// SIMATIC S7-200 project (STEP 7-Micro/WIN), CPU 224XP CN REL 02.02

SYMBOL_TABLE 用户定义3
一楼呼叫             I0.1     // SB1
二楼呼叫             I0.2     // SB2
三楼呼叫             I0.3     // SB3
响应一楼呼叫           Q0.1     // HL1
响应二楼呼叫           Q0.2     // HL2
响应三楼呼叫           Q0.3     // HL3
一楼响应保持           M1.1
二楼响应保持           M1.2
三楼响应保持           M1.3
电梯在一楼            Q0.4     // SQ1
电梯在二楼            Q0.5     // SQ2
电梯在三楼            Q0.6     // SQ3
开门               Q0.0
关门               Q2.1
电梯停止             Q0.7
电机正转             Q1.0     // 正在上升
电机反转             Q1.1     // 下降
上升保持             M3.2     // 电梯属于上升状态
下降保持             M3.3     // 电梯属于下降状态
楼层位置             VW0      // 数据寄存，1楼值1，2楼值2
呼叫数              VW2      // 有多少个电梯正在呼叫
上行定时器            T37      // 电梯移动时间的计数器
下行定时器            T38
开始关门             T56
停止关门             T57
门寄存器             M2.0     // 前4秒开门灯亮，第4秒关灯亮，第5秒继续运行
重置               I0.0     // 按下后电梯重置
END_SYMBOL_TABLE

ORGANIZATION_BLOCK 主程序:OB1
TITLE=程序注释
BEGIN
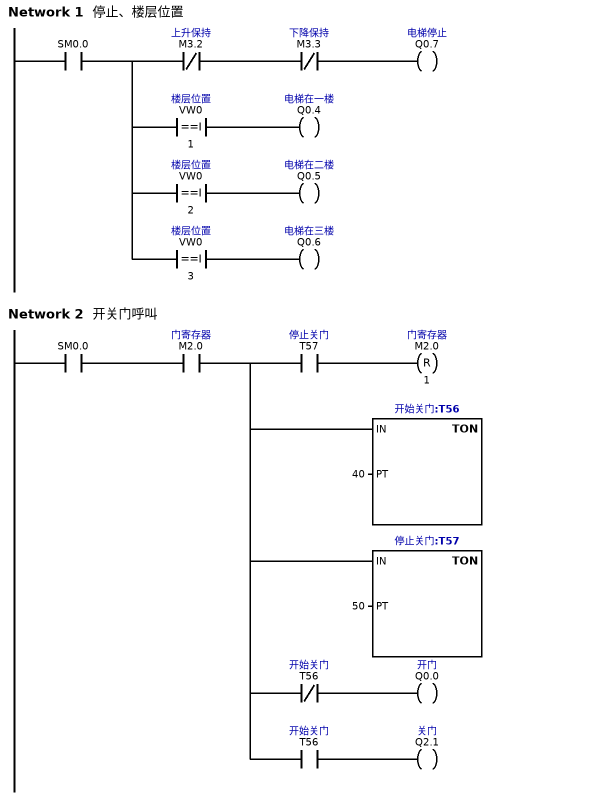
Network 1 // 停止、楼层位置
LD     SM0.0
LPS
AN     上升保持:M3.2
AN     下降保持:M3.3
=      电梯停止:Q0.7
LRD
AW=    楼层位置:VW0, 1
=      电梯在一楼:Q0.4
LRD
AW=    楼层位置:VW0, 2
=      电梯在二楼:Q0.5
LPP
AW=    楼层位置:VW0, 3
=      电梯在三楼:Q0.6
Network 2 // 开关门呼叫
LD     SM0.0
A      门寄存器:M2.0
LPS
A      停止关门:T57
R      门寄存器:M2.0, 1
LRD
TON    开始关门:T56, 40
LRD
TON    停止关门:T57, 50
LRD
AN     开始关门:T56
=      开门:Q0.0
LPP
A      开始关门:T56
=      关门:Q2.1
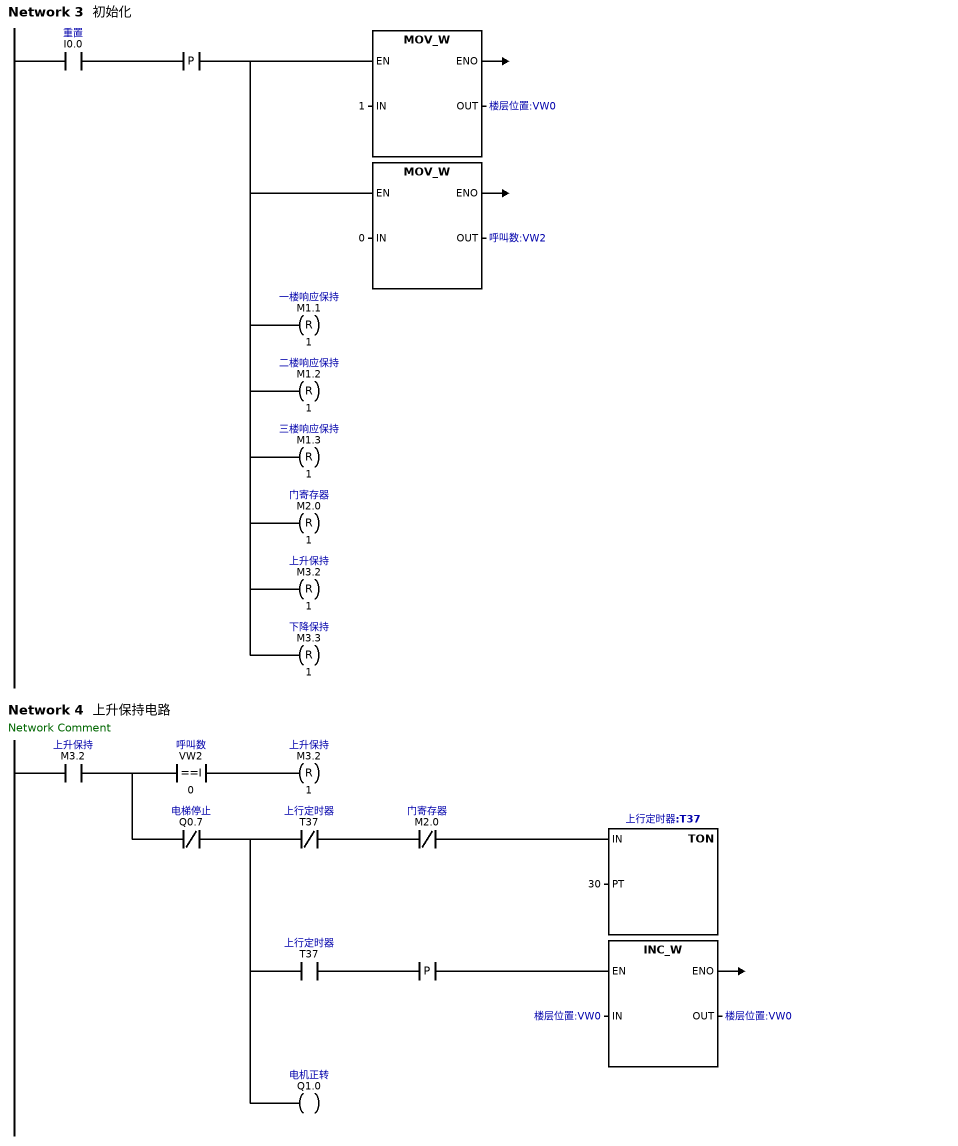
Network 3 // 初始化
LD     重置:I0.0
EU
MOVW   1, 楼层位置:VW0
MOVW   0, 呼叫数:VW2
R      一楼响应保持:M1.1, 1
R      二楼响应保持:M1.2, 1
R      三楼响应保持:M1.3, 1
R      门寄存器:M2.0, 1
R      上升保持:M3.2, 1
R      下降保持:M3.3, 1
Network 4 // 上升保持电路
// Network Comment
LD     上升保持:M3.2
LPS
AW=    呼叫数:VW2, 0
R      上升保持:M3.2, 1
LPP
AN     电梯停止:Q0.7
LPS
AN     上行定时器:T37
AN     门寄存器:M2.0
TON    上行定时器:T37, 30
LRD
A      上行定时器:T37
EU
INCW   楼层位置:VW0
LPP
=      电机正转:Q1.0
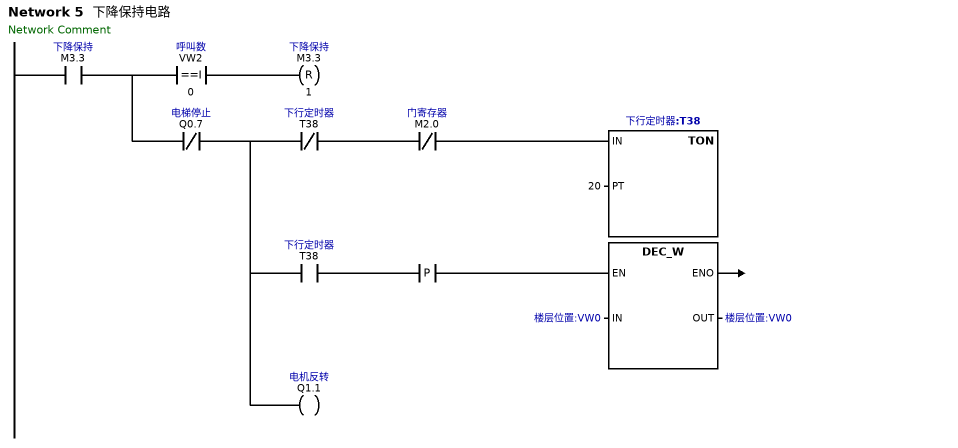
Network 5 // 下降保持电路
// Network Comment
LD     下降保持:M3.3
LPS
AW=    呼叫数:VW2, 0
R      下降保持:M3.3, 1
LPP
AN     电梯停止:Q0.7
LPS
AN     下行定时器:T38
AN     门寄存器:M2.0
TON    下行定时器:T38, 20
LRD
A      下行定时器:T38
EU
DECW   楼层位置:VW0
LPP
=      电机反转:Q1.1
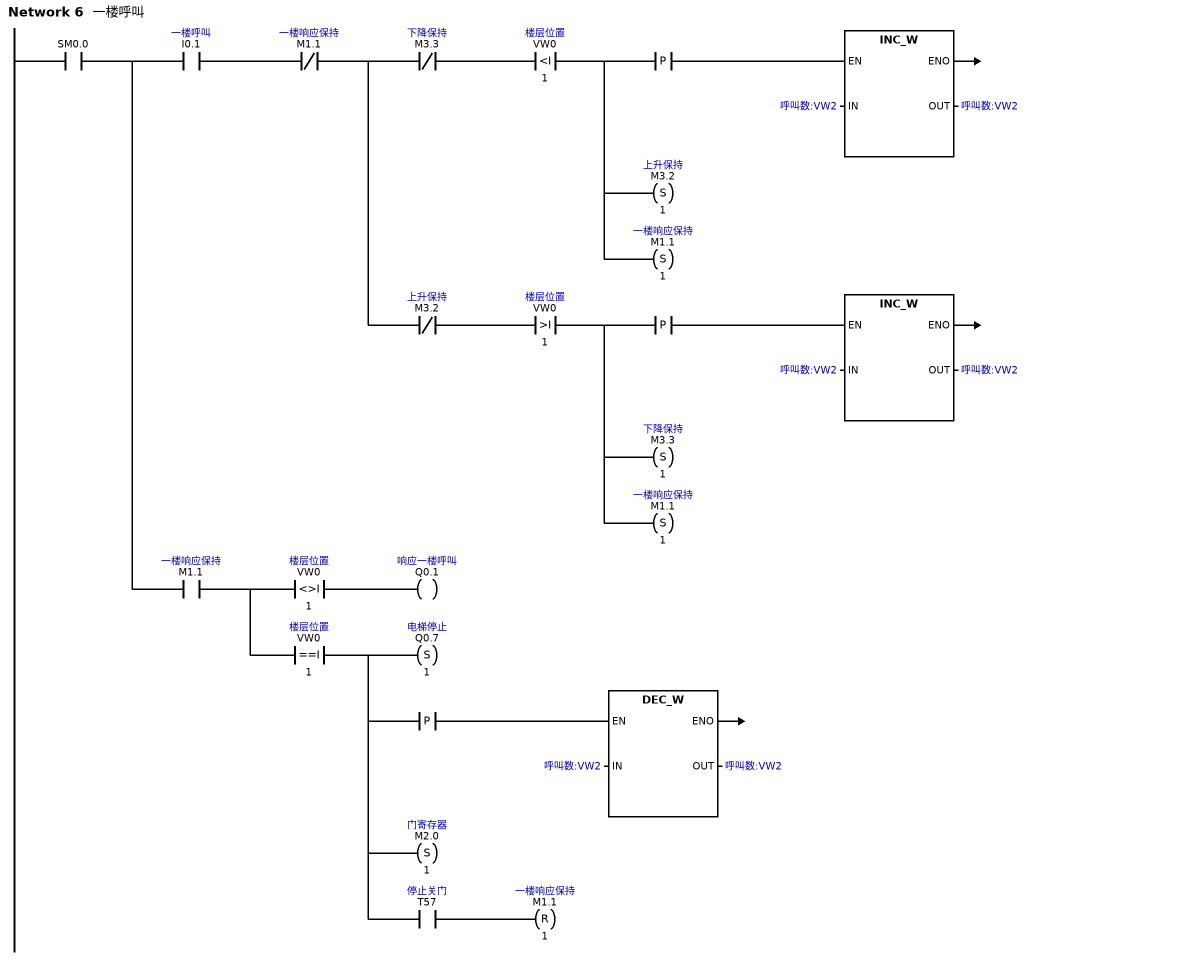
Network 6 // 一楼呼叫
LD     SM0.0
LPS
A      一楼呼叫:I0.1
AN     一楼响应保持:M1.1
LPS
AN     下降保持:M3.3
AW<    楼层位置:VW0, 1
LPS
EU
INCW   呼叫数:VW2
LRD
S      上升保持:M3.2, 1
LPP
S      一楼响应保持:M1.1, 1
LPP
AN     上升保持:M3.2
AW>    楼层位置:VW0, 1
LPS
EU
INCW   呼叫数:VW2
LRD
S      下降保持:M3.3, 1
LPP
S      一楼响应保持:M1.1, 1
LPP
A      一楼响应保持:M1.1
LPS
AW<>   楼层位置:VW0, 1
=      响应一楼呼叫:Q0.1
LPP
AW=    楼层位置:VW0, 1
LPS
S      电梯停止:Q0.7, 1
EU
DECW   呼叫数:VW2
LRD
S      门寄存器:M2.0, 1
LPP
A      停止关门:T57
R      一楼响应保持:M1.1, 1
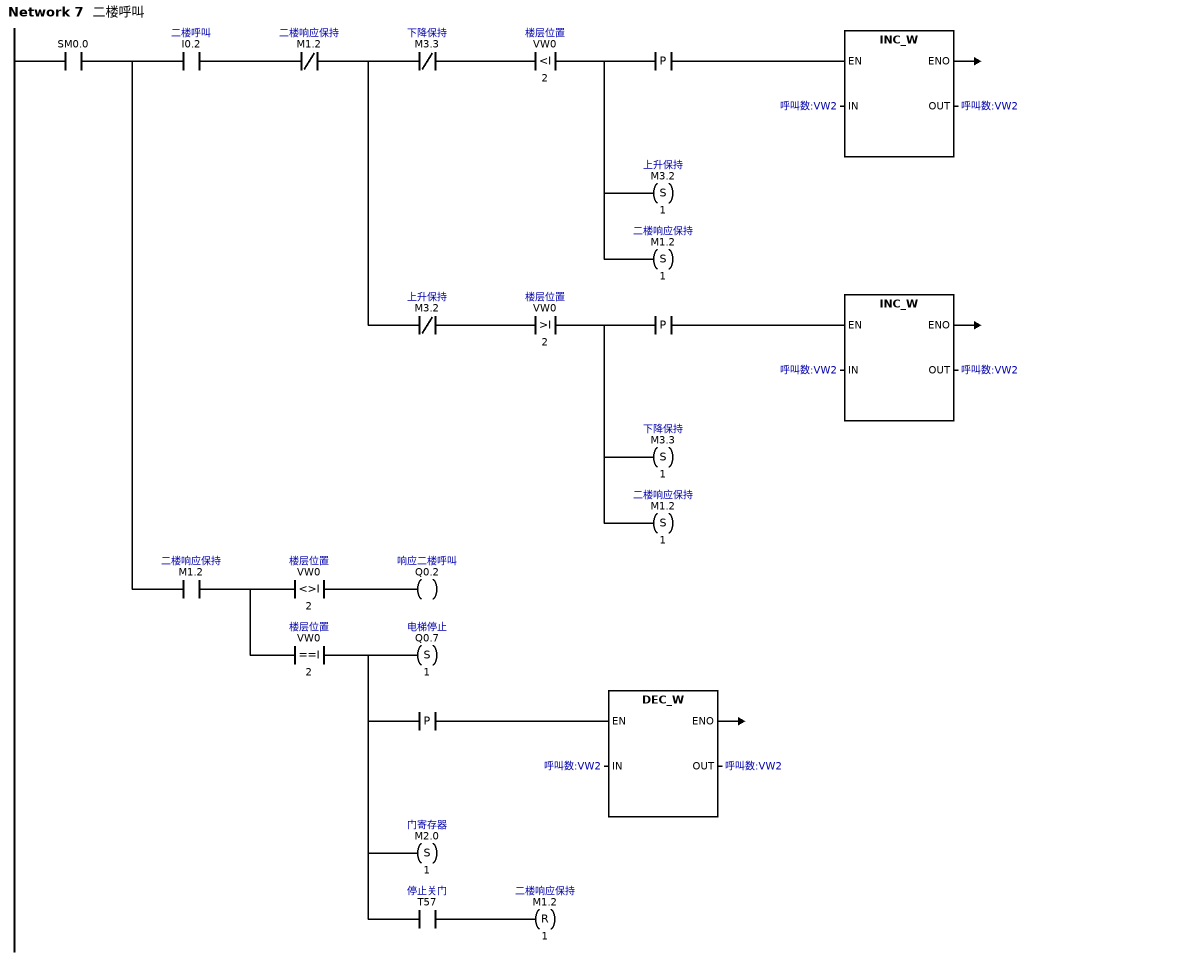
Network 7 // 二楼呼叫
LD     SM0.0
LPS
A      二楼呼叫:I0.2
AN     二楼响应保持:M1.2
LPS
AN     下降保持:M3.3
AW<    楼层位置:VW0, 2
LPS
EU
INCW   呼叫数:VW2
LRD
S      上升保持:M3.2, 1
LPP
S      二楼响应保持:M1.2, 1
LPP
AN     上升保持:M3.2
AW>    楼层位置:VW0, 2
LPS
EU
INCW   呼叫数:VW2
LRD
S      下降保持:M3.3, 1
LPP
S      二楼响应保持:M1.2, 1
LPP
A      二楼响应保持:M1.2
LPS
AW<>   楼层位置:VW0, 2
=      响应二楼呼叫:Q0.2
LPP
AW=    楼层位置:VW0, 2
LPS
S      电梯停止:Q0.7, 1
EU
DECW   呼叫数:VW2
LRD
S      门寄存器:M2.0, 1
LPP
A      停止关门:T57
R      二楼响应保持:M1.2, 1
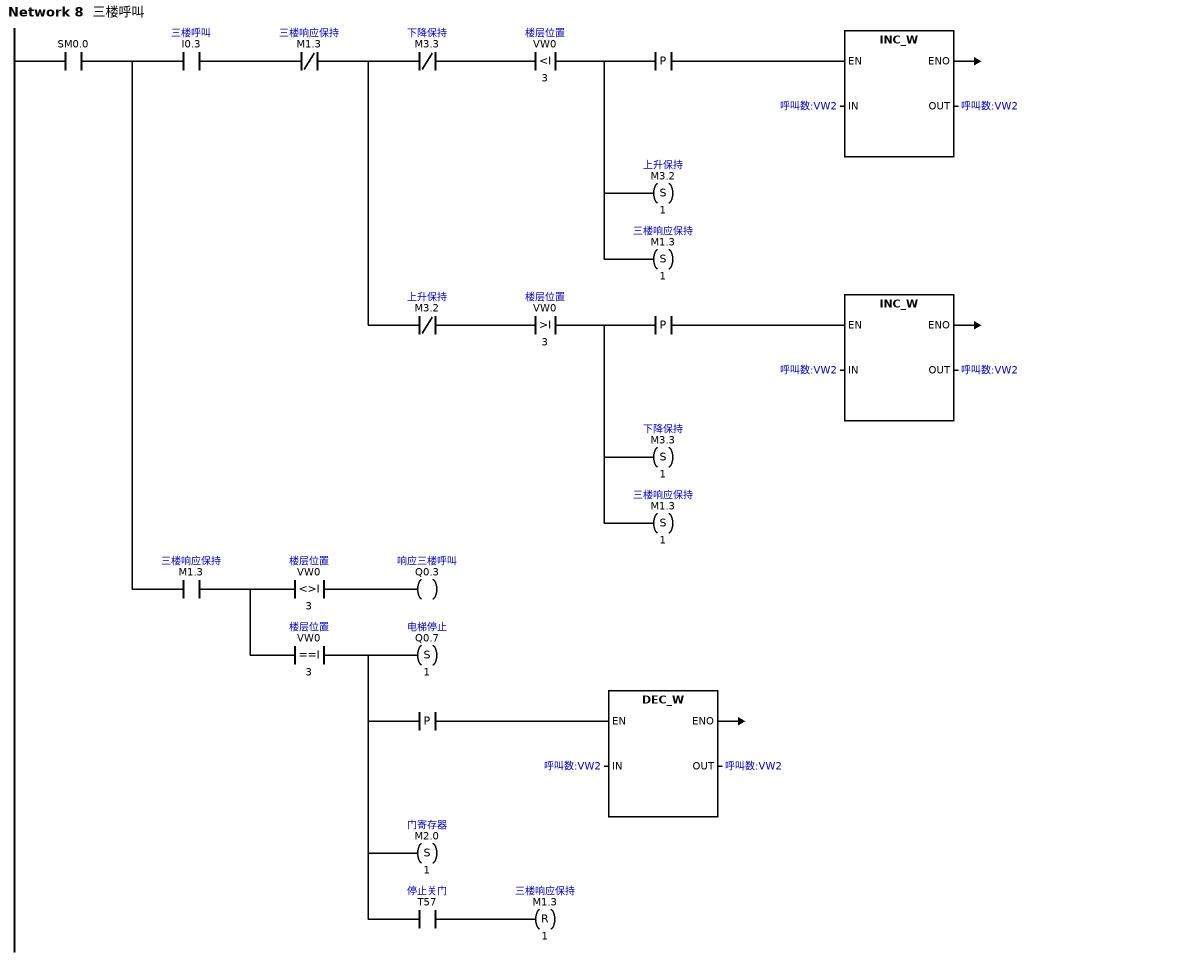
Network 8 // 三楼呼叫
LD     SM0.0
LPS
A      三楼呼叫:I0.3
AN     三楼响应保持:M1.3
LPS
AN     下降保持:M3.3
AW<    楼层位置:VW0, 3
LPS
EU
INCW   呼叫数:VW2
LRD
S      上升保持:M3.2, 1
LPP
S      三楼响应保持:M1.3, 1
LPP
AN     上升保持:M3.2
AW>    楼层位置:VW0, 3
LPS
EU
INCW   呼叫数:VW2
LRD
S      下降保持:M3.3, 1
LPP
S      三楼响应保持:M1.3, 1
LPP
A      三楼响应保持:M1.3
LPS
AW<>   楼层位置:VW0, 3
=      响应三楼呼叫:Q0.3
LPP
AW=    楼层位置:VW0, 3
LPS
S      电梯停止:Q0.7, 1
EU
DECW   呼叫数:VW2
LRD
S      门寄存器:M2.0, 1
LPP
A      停止关门:T57
R      三楼响应保持:M1.3, 1
END_ORGANIZATION_BLOCK
